(* IEC 61131-3 sources: axftcmlib/test, 13 files *)

(* ---- ActuatorTimeBasedTest.st ---- *)
USING Simatic.Ax.Commands;
USING Simatic.Ax.axftcmlib;
USING Simatic.Ax.IO.Output;
USING AxUnit.Assert;

NAMESPACE Simatic.Ax.axftcmlib

    {TestFixture}
    CLASS ActuatorTimeBasedTest
        VAR PROTECTED
            _actuator : ActuatorTimeBased;
            _actuatorStateLess : ActuatorTimeBased;
            _output : BinOutput;
            cmd : itfCommand;
            busy : BOOL;
        END_VAR

        {TestSetup}
        METHOD PUBLIC SetUp
            _actuator := _actuatorStateLess;
            _actuator.Q_ToWorkPosition := _output;
        END_METHOD

                {Test}
        METHOD PUBLIC TestTurnPneumaticCylinderPush_Expect_state_is_On
            cmd := _actuator.GoToWorkPosition();
            busy := cmd.Busy();
            AxUnit.Assert.Equal(expected := TRUE, actual := busy);
            AxUnit.Assert.Equal(expected := TRUE, actual := _output.IsOn());
            Equal(expected := TRUE, actual := _actuator.GetState() = ActuatorState#InWorkPosition);
        END_METHOD

        {Test}
        METHOD PUBLIC TestZylinderNotAsigned_Expected_ErrorFound_is_True
            VAR
                Test : BOOL;
            END_VAR
            _actuator.Q_ToWorkPosition := NULL;
            _actuator.Busy();
            AxUnit.Assert.Equal(Expected := TRUE, actual := _actuator.Error());
            ;
        END_METHOD

        {Test}
        METHOD PUBLIC TestPneumaticCylinderError_Expected_ErrorFound_TRUE
            VAR
                Test : BOOL;
            END_VAR

            Test := _actuator.Error();
            AxUnit.Assert.Equal(Expected := FALSE, actual := Test);
            ;
        END_METHOD

    END_CLASS

END_NAMESPACE

(* ---- Axis_Mock.st ---- *)
USING Simatic.Ax.IO.Input;
USING System.Timer;
USING Simatic.Ax.SimpleControlModules;

NAMESPACE Simatic.Ax.axftcmlib
    CLASS Axis_Mock
        IMPLEMENTS IAxis
        VAR PUBLIC
            State : PlcOpenState;
        END_VAR
        VAR PROTECTED

        END_VAR

        //-----------------------------------------
        // interface implementation
        METHOD PUBLIC MoveVelocity
            VAR_INPUT
                velocity : LREAL;
                direction : Direction;
            END_VAR
            ;
        END_METHOD
        METHOD PUBLIC MoveRelative : BOOL
            VAR_INPUT
                velocity : LREAL;
                distance : LINT;
            END_VAR
;
        END_METHOD
        METHOD PUBLIC MoveAbsolute : BOOL
            VAR_INPUT
                velocity : LREAL;
                position : LINT;
            END_VAR
;
        END_METHOD
        METHOD PUBLIC Homing : BOOL
            VAR_INPUT
                velocity : LREAL;
                direction : Direction;
            END_VAR
;
        END_METHOD
        METHOD PUBLIC Halt
            ;
        END_METHOD
        METHOD PUBLIC IsHomed : BOOL
            ;
        END_METHOD

        //-------------------------------------------------------------------------------
        // Section for private methods

        METHOD PUBLIC IsRunning : BOOL
            IsRunning := State = PlcOpenstate#Busy;
        END_METHOD

        METHOD PUBLIC Homing : BOOL
            VAR_INPUT
                Position : LINT;
            END_VAR

            ;
        END_METHOD
END_CLASS

END_NAMESPACE

(* ---- ColorSensor_test.st ---- *)
USING AxUnit.Assert;

NAMESPACE Simatic.Ax.axftcmlib
    {TestFixture}
    Class MyColorSensorTest

        VAR PROTECTED
            _testColorSensor : ColorSensor;
            //_testSubject : colors;
        END_VAR

        // METHOD PROTECTED SetUp
        //     _testColorSensor.OutputColor := _testSubject;
        // END_METHOD

        {Test}
        METHOD PUBLIC TestDetectionWhite_Expect_True
            VAR_TEMP
                Dummy : BOOL;
            END_VAR

            // THIS.SetUp();
            Dummy := FALSE;
            _testColorSensor.detectColor(DetectedColorValue := 9000);
            IF _testColorSensor.OutputColor = 1 THEN
                Dummy := TRUE;
            END_IF;
            AxUnit.Assert.Equal(expected := TRUE, actual := Dummy);
        END_METHOD

        {Test}
        METHOD PUBLIC TestDetectionRed_Expect_True
            VAR_TEMP
                Dummy : BOOL;
            END_VAR

            // THIS.SetUp();
            Dummy := FALSE;
            _testColorSensor.detectColor(DetectedColorValue := 14000);
            IF _testColorSensor.OutputColor = 2 THEN
                Dummy := TRUE;
            END_IF;
            AxUnit.Assert.Equal(expected := TRUE, actual := Dummy);
        END_METHOD

        {Test}
        METHOD PUBLIC TestDetectionBlue_Expect_True
            VAR_TEMP
                Dummy : BOOL;
            END_VAR

            // THIS.SetUp();
            Dummy := FALSE;
            _testColorSensor.detectColor(DetectedColorValue := 19000);
            IF _testColorSensor.OutputColor = 3 THEN
                Dummy := TRUE;
            END_IF;
            AxUnit.Assert.Equal(expected := TRUE, actual := Dummy);
        END_METHOD

    END_CLASS
END_NAMESPACE

(* ---- Compressor_test.st ---- *)
//USING Simatic.Ax.Cylinder;
USING AxUnit.Assert;
USING Simatic.Ax.IO.Input;
USING Simatic.Ax.axftcmlib;
USING Simatic.Ax.IO.Output;

NAMESPACE Simatic.Ax.axftcmlib
    {TestFixture}
    CLASS MyCompressorTest
        VAR PROTECTED
            _testCompressor : PneumaticCompressor;
            _testSubject : BinOutput;
        END_VAR
        METHOD PUBLIC  SetUp
            _testCompressor.ActiveCompressor := _testSubject;
        END_METHOD

        {Test}
        METHOD PUBLIC TestTurnCompressorOn_Expect_state_is_On
            THIS.SetUp();
            _testCompressor.PneumaticCompressorOn();
            AxUnit.Assert.Equal(expected := TRUE, actual :=_testSubject.IsOn()); // _testCompressor.ActiveCompressor.IsOn());
        END_METHOD

        {Test}
        METHOD PUBLIC TestTurnCompressorOff_Expect_state_is_Off
            THIS.SetUp();
            _testCompressor.PneumaticCompressorOff();
            AxUnit.Assert.Equal(expected := FALSE, actual := _testSubject.IsOn());
            END_METHOD

    END_CLASS
END_NAMESPACE

(* ---- Encoder_test.st ---- *)
USING Simatic.Ax.axftcmlib;

NAMESPACE Simatic.Ax.axftcmlib

    {TestFixture}
    CLASS MyEncoderTest
        VAR PROTECTED
            _testEncoderStatic : TimeBasedEncoder;
            _staticTimeProvider : TimeProviderMOCK_100ms_const;
            _staticAxis : Axis_Mock := (State := PlcOpenState#Busy);
        END_VAR

        METHOD PUBLIC SetUp
            VAR
                velocity : LREAL;
                dummyValue : INT;
            END_VAR
            dummyValue := 0;
            velocity := 1.0;
            _testEncoderStatic.velocity := 1.0;
            _testEncoderStatic.TimeProvider := _staticTimeProvider;
            _testEncoderStatic.EncoderAxis := _staticAxis;
            _testEncoderStatic.EncoderAxis.MoveVelocity(velocity, dummyvalue);
        END_METHOD

        {Test}
        METHOD PUBLIC TestPositionAfter100ms_Expect_position_equal
            THIS.SetUp();
            _testEncoderStatic.Reset();
            _testEncoderStatic.Evaluate();
            AxUnit.Assert.Equal(expected := 100, actual := _testEncoderStatic.GetValue());
            _testEncoderStatic.Evaluate();
            AxUnit.Assert.Equal(expected := 200, actual := _testEncoderStatic.GetValue());
            // Set Axis to stop
            _staticAxis.State := PlcOpenState#Done;
            _testEncoderStatic.Evaluate();
            AxUnit.Assert.Equal(expected := 200, actual := _testEncoderStatic.GetValue()); // dont integrate when axis is stopped
            // After Reset the GetValue should be 0
            _testEncoderStatic.Reset();
            AxUnit.Assert.Equal(expected := 0, actual := _testEncoderStatic.GetValue());

        END_METHOD
    END_CLASS

END_NAMESPACE

(* ---- test.st ---- *)
USING Simatic.Ax.IO.Input;
USING Simatic.Ax.Commands;
USING Simatic.Ax.axftcmlib;
USING Simatic.Ax.IO.Output;
USING AxUnit.Assert;

NAMESPACE Simatic.Ax.axftcmlib

    {TestFixture}
    CLASS TwoWayActuatorTest
        VAR PROTECTED
            _actuator : TwoWayActuator;
            _actuatorStateLess : TwoWayActuator;
            _qToWork : BinOutput;
            _qToHome : BinOutput;
            _outputStateLess : BinOutput;
            _iInHomePos : BinSignal;
            _iInWorkPos : BinSignal;
            _binSignalStateless : BinSignal;
            cmd : itfCommand;
            done : BOOL;
            busy : BOOL;
        END_VAR

        {TestSetup}
        METHOD PUBLIC SetUp
            _actuator := _actuatorStateLess;
            _actuator.Q_ToWorkPosition := _qToWork;
            _actuator.Q_ToHomePosition := _qToHome;
            _actuator.I_InHomePosition := _iInHomePos;
            _actuator.I_InWorkPosition := _iInWorkPos;
            _iInHomePos := _binSignalStateless;
            _iInWorkPos := _binSignalStateless;
            _qToWork := _outputStateLess;
            _qToHome := _outputStateLess;
            busy := FALSE;
            cmd := NULL;
        END_METHOD

        {Test}
        METHOD PUBLIC GoToWorkPosition_Swiches_Q_ToWorkPosition_On_And_Returns_Busy
            cmd := _actuator.GoToWorkPosition();
            busy := cmd.Busy();
            AxUnit.Assert.Equal(expected := TRUE, actual := busy);
            AxUnit.Assert.Equal(expected := TRUE, actual := _qToWork.IsOn());
            AxUnit.Assert.Equal(expected := FALSE, actual := _qToHome.IsOn());
            Equal(expected := TRUE, actual := _actuator.GetState() = ActuatorState#MoveToWorkPosition);
        END_METHOD

        {Test}
        METHOD PUBLIC GoToWorkPosition_Returns_Done_When_end_position_is_already_reached
            _iInWorkPos.ReadCyclic(signal := TRUE);
            cmd := _actuator.GoToWorkPosition();
            busy := cmd.Busy();
            IF NOT(busy) THEN
                done := cmd.Done();
            END_IF;
            AxUnit.Assert.Equal(expected := FALSE, actual := busy);
            AxUnit.Assert.Equal(expected := TRUE, actual := done);
            AxUnit.Assert.Equal(expected := FALSE, actual := _qToWork.IsOn());
            AxUnit.Assert.Equal(expected := FALSE, actual := _qToHome.IsOn());
            Equal(expected := TRUE, actual := _actuator.GetState() = ActuatorState#InWorkPosition);
        END_METHOD

        {Test}
        METHOD PUBLIC Reaching_WorkPosition_Switches_Q_ToWorkPosition_Off_And_Returns_Done
            THIS.GoToWorkPosition_Swiches_Q_ToWorkPosition_On_And_Returns_Busy();
            _iInWorkPos.ReadCyclic(signal := TRUE);
            busy := cmd.Busy();
            IF NOT(busy) THEN
                done := cmd.Done();
            END_IF;
            AxUnit.Assert.Equal(expected := FALSE, actual := busy);
            AxUnit.Assert.Equal(expected := TRUE, actual := done);
            AxUnit.Assert.Equal(expected := FALSE, actual := _qToWork.IsOn());
            AxUnit.Assert.Equal(expected := FALSE, actual := _qToHome.IsOn());
            Equal(expected := TRUE, actual := _actuator.GetState() = ActuatorState#InWorkPosition);
        END_METHOD

        // Test Home Position
        {Test}
        METHOD PUBLIC GoToHomePosition_Swiches_Q_ToHomePosition_On_And_Returns_Busy
            cmd := _actuator.GoToHomePosition();
            busy := cmd.Busy();
            AxUnit.Assert.Equal(expected := TRUE, actual := busy);
            AxUnit.Assert.Equal(expected := FALSE, actual := _qToWork.IsOn());
            AxUnit.Assert.Equal(expected := TRUE, actual := _qToHome.IsOn());
            Equal(expected := TRUE, actual := _actuator.GetState() = ActuatorState#MoveToHomePosition);
        END_METHOD

        {Test}
        METHOD PUBLIC GoToHomePosition_Returns_Done_When_end_position_is_already_reached
            _iInHomePos.ReadCyclic(signal := TRUE);
            cmd := _actuator.GoToHomePosition();
            busy := cmd.Busy();
            IF NOT(busy) THEN
                done := cmd.Done();
            END_IF;
            AxUnit.Assert.Equal(expected := FALSE, actual := busy);
            AxUnit.Assert.Equal(expected := TRUE, actual := done);
            AxUnit.Assert.Equal(expected := FALSE, actual := _qToWork.IsOn());
            AxUnit.Assert.Equal(expected := FALSE, actual := _qToHome.IsOn());
            Equal(expected := TRUE, actual := _actuator.GetState() = ActuatorState#InHomePosition);
        END_METHOD

        {Test}
        METHOD PUBLIC Reaching_HomePosition_Switches_Q_ToHomePosition_Off_And_Returns_Done
            THIS.GoToHomePosition_Swiches_Q_ToHomePosition_On_And_Returns_Busy();
            _iInHomePos.ReadCyclic(signal := TRUE);
            busy := cmd.Busy();
            IF NOT(busy) THEN
                done := cmd.Done();
            END_IF;
            AxUnit.Assert.Equal(expected := FALSE, actual := busy);
            AxUnit.Assert.Equal(expected := TRUE, actual := done);
            AxUnit.Assert.Equal(expected := FALSE, actual := _qToWork.IsOn());
            AxUnit.Assert.Equal(expected := FALSE, actual := _qToHome.IsOn());
            Equal(expected := TRUE, actual := _actuator.GetState() = ActuatorState#InHomePosition);
        END_METHOD
    END_CLASS

END_NAMESPACE

(* ---- TestAxis.st ---- *)
USING Simatic.Ax.IO.Output;
USING Simatic.Ax.IO.Input;
USING Simatic.Ax.axftcmlib;
USING AxUnit.Assert;

// USING Simatic.Ax.SimpleControlModules;
NAMESPACE Simatic.Ax.Library

    {TestFixture}
    CLASS TestAxisHoming
        VAR PROTECTED
            _axis : Axis;
            _refSwitch : BinSignal;
            _motor : MotorFT;
            _fwd : BinOutput;
            _rvs : BinOutput;
            _encoder : Simatic.Ax.SimpleControlModules.EncoderAB;
        END_VAR
        METHOD PUBLIC Setup
            _motor.Forward := _fwd;
            _motor.Reverse := _rvs;
            _axis.Motor := _motor;
            _axis.Encoder := _encoder;
            _axis.ReferenceSwitch := _refSwitch;
        END_METHOD
        {Test}
        METHOD PUBLIC TestForwardDirection_Expect_Fwd_IsOn
            THIS.Setup();
            _axis.MoveVelocity(direction := Direction#Forward);
            _axis.RunCyclic();
            Equal(expected := TRUE, actual := _axis.GetPlcOpenState() = PlcOpenState#Busy);
            Equal(expected := TRUE, actual := _fwd.IsOn());
            Equal(expected := FALSE, actual := _rvs.IsOn());
        END_METHOD
        {Test}
        METHOD PUBLIC Homing_from_outside_of_the_referecne_sensor_Move_reverse
            THIS.Setup();
            _axis.Homing(direction := Direction#Reverse);
            _axis.RunCyclic();
            Equal(expected := TRUE, actual := _axis.GetPlcOpenState() = PlcOpenState#Busy);
            _axis.RunCyclic();
            Equal(expected := FALSE, actual := _fwd.IsOn());
            Equal(expected := TRUE, actual := _rvs.IsOn());
        END_METHOD

        {Test}
        METHOD PUBLIC Homing_from_outside_of_the_referecne_sensor_Move_forward
            THIS.Setup();
            _axis.Homing(direction := Direction#Forward);
            _axis.RunCyclic();
            Equal(expected := TRUE, actual := _axis.GetPlcOpenState() = PlcOpenState#Busy);
            _axis.RunCyclic();
            Equal(expected := TRUE, actual := _fwd.IsOn());
            Equal(expected := FALSE, actual := _rvs.IsOn());
        END_METHOD

        {Test}
        METHOD PUBLIC Homing_untilsensor_has_reached
            VAR_TEMP
                isHomed : BOOL;
            END_VAR
            THIS.Setup();

            _axis.Homing(direction := Direction#Forward);
            _axis.RunCyclic();

            _refSwitch.ReadCyclic(signal := FALSE);
            _axis.RunCyclic();
            Equal(expected := TRUE, actual := _axis.GetPlcOpenState() = PlcOpenState#Busy);
            Equal(expected := FALSE, actual := _axis.GetPlcOpenState() = PlcOpenState#Error);
            Equal(expected := FALSE, actual := _axis.GetPlcOpenState() = PlcOpenState#Done);
            Equal(expected := TRUE, actual := _fwd.IsOn());
            Equal(expected := FALSE, actual := _rvs.IsOn());

            _refSwitch.ReadCyclic(signal := FALSE);
            _axis.RunCyclic();
            Equal(expected := TRUE, actual := _axis.GetPlcOpenState() = PlcOpenState#Busy);
            Equal(expected := FALSE, actual := _axis.GetPlcOpenState() = PlcOpenState#Error);
            Equal(expected := FALSE, actual := _axis.GetPlcOpenState() = PlcOpenState#Done);
            Equal(expected := TRUE, actual := _fwd.IsOn());
            Equal(expected := FALSE, actual := _rvs.IsOn());

            _refSwitch.ReadCyclic(signal := FALSE);
            _axis.RunCyclic();
            Equal(expected := TRUE, actual := _axis.GetPlcOpenState() = PlcOpenState#Busy);
            Equal(expected := FALSE, actual := _axis.GetPlcOpenState() = PlcOpenState#Error);
            Equal(expected := FALSE, actual := _axis.GetPlcOpenState() = PlcOpenState#Done);
            Equal(expected := TRUE, actual := _fwd.IsOn());
            Equal(expected := FALSE, actual := _rvs.IsOn());

            _refSwitch.ReadCyclic(signal := TRUE);
            _axis.RunCyclic();
            _axis.RunCyclic();
            Equal(expected := FALSE, actual := _axis.GetPlcOpenState() = PlcOpenState#Busy);
            Equal(expected := FALSE, actual := _axis.GetPlcOpenState() = PlcOpenState#Error);
            Equal(expected := TRUE, actual := _axis.GetPlcOpenState() = PlcOpenState#Done);
            Equal(expected := FALSE, actual := _fwd.IsOn());
            Equal(expected := FALSE, actual := _rvs.IsOn());
            Equal(expected := TRUE, actual := _axis.IsHomed());
        END_METHOD

    END_CLASS

END_NAMESPACE

(* ---- TestAxisManualHoming.st ---- *)
USING Simatic.Ax.IO.Output;
USING Simatic.Ax.IO.Input;
USING Simatic.Ax.axftcmlib;
USING AxUnit.Assert;

// USING Simatic.Ax.SimpleControlModules;
NAMESPACE Simatic.Ax.Library

    {TestFixture}
    CLASS TestAxisManualHoming
        VAR PROTECTED
            _axis : Axis;
            _refSwitch : BinSignal;
            _motor : MotorFT;
            _fwd : BinOutput;
            _rvs : BinOutput;
            _encoder : Simatic.Ax.SimpleControlModules.EncoderAB;
        END_VAR
        METHOD PUBLIC Setup
            _motor.Forward := _fwd;
            _motor.Reverse := _rvs;
            _axis.Motor := _motor;
            _axis.Encoder := _encoder;
            _axis.ReferenceSwitch := _refSwitch;
        END_METHOD
        {Test}
        METHOD PUBLIC AxisReturnes_IsHomed_when_Homing_Method_isCalled
            THIS.Setup();
            Equal(expected := FALSE, actual := _axis.IsHomed());
            _axis.Homing(position := 100);
            Equal(expected := TRUE, actual := _axis.IsHomed());
            Equal(expected := TRUE, actual := _axis.GetPlcOpenState() = PlcOpenState#Done);
            _axis.RunCyclic();
            Equal(expected := FALSE, actual := _axis.GetPlcOpenState() = PlcOpenState#Done);
        END_METHOD
    END_CLASS

END_NAMESPACE

(* ---- TestAxisMoveAbsolut.st ---- *)
USING Simatic.Ax.IO.Output;
USING Simatic.Ax.IO.Input;
USING Simatic.Ax.axftcmlib;
USING AxUnit.Assert;

// USING Simatic.Ax.SimpleControlModules;
NAMESPACE Simatic.Ax.Library

    {TestFixture}
    CLASS TestAxisMoveAbsolut
        VAR PROTECTED
            _axis : Axis;
            _refSwitch : BinSignal;
            _motor : MotorFT;
            _fwd : BinOutput;
            _rvs : BinOutput;
            _encoder : Simatic.Ax.SimpleControlModules.EncoderAB;
        END_VAR
        METHOD PUBLIC Setup
            _motor.Forward := _fwd;
            _motor.Reverse := _rvs;
            _axis.Motor := _motor;
            _axis.Encoder := _encoder;
            _axis.ReferenceSwitch := _refSwitch;
        END_METHOD
        METHOD PUBLIC Home : BOOL
            VAR_INPUT
                axis : REF_TO Axis;
                refSwitch : REF_TO BinSignal;
            END_VAR
            axis^.Homing(direction := Direction#Forward);
            refSwitch^.ReadCyclic(signal := FALSE);
            axis^.RunCyclic();
            refSwitch^.ReadCyclic(signal := TRUE);
            axis^.RunCyclic();
            // one additional cycle to finalize the Homing
            axis^.RunCyclic();
            Home := axis^.IsHomed();
        END_METHOD
        {Test}
        METHOD PUBLIC Test_MoveAbsolut_on_a_not_homed_axis_which_results_in_an_error
            VAR_TEMP
                isHomed : BOOL;
            END_VAR
            THIS.Setup();
            _axis.MoveAbsolute(velocity := 100.0, position := LINT#100);
            _axis.RunCyclic();
            Equal(expected := FALSE, actual := _axis.GetPlcOpenState() = PlcOpenState#Busy);
            Equal(expected := TRUE, actual := _axis.GetPlcOpenState() = PlcOpenState#Error);
            Equal(expected := FALSE, actual := _axis.GetPlcOpenState() = PlcOpenState#Done);
        END_METHOD
        {Test}
        METHOD PUBLIC Test_MoveAbsolut_on_a_homed_axis
            VAR_TEMP
                isHomed : BOOL;
            END_VAR
            THIS.Setup();
            isHomed := THIS.Home(axis := REF(_axis), refSwitch := REF(_refSwitch));
            Equal(expected := TRUE, actual := isHomed);
            Equal(expected := FALSE, actual := _fwd.IsOn());
            Equal(expected := FALSE, actual := _rvs.IsOn());
            // start Axis to move to position 100
            _axis.MoveAbsolute(velocity := 100.0, position := LINT#100);
            _axis.RunCyclic();
            Equal(expected := TRUE, actual := _axis.GetPlcOpenState() = PlcOpenState#Busy);
            Equal(expected := FALSE, actual := _axis.GetPlcOpenState() = PlcOpenState#Error);
            Equal(expected := FALSE, actual := _axis.GetPlcOpenState() = PlcOpenState#Done);
            Equal(expected := TRUE, actual := _fwd.IsOn());
            Equal(expected := FALSE, actual := _rvs.IsOn());
            // Axis is at position 99
            _encoder.SetValue(value := LINT#99);
            _axis.RunCyclic();
            Equal(expected := TRUE, actual := _axis.GetPlcOpenState() = PlcOpenState#Busy);
            // test axis in position
            _encoder.SetValue(value := LINT#100);
            _axis.RunCyclic();
            _axis.RunCyclic();
            Equal(expected := TRUE, actual := _axis.GetPlcOpenState() = PlcOpenState#Done);
            Equal(expected := FALSE, actual := _axis.GetPlcOpenState() = PlcOpenState#Busy);
            Equal(expected := FALSE, actual := _fwd.IsOn());
            Equal(expected := FALSE, actual := _rvs.IsOn());            // test axis in position - done after one cycle is false
            _encoder.SetValue(value := LINT#100);
            _axis.RunCyclic();
            Equal(expected := FALSE, actual := _axis.GetPlcOpenState() = PlcOpenState#Done);
            Equal(expected := FALSE, actual := _axis.GetPlcOpenState() = PlcOpenState#Busy);
        END_METHOD
        {Test}
        METHOD PUBLIC Move_Absolut_on_a_axis_which_is_already_inPos
            VAR_TEMP
                isHomed : BOOL;
            END_VAR
            THIS.Setup();
            isHomed := THIS.Home(axis := REF(_axis), refSwitch := REF(_refSwitch));
            Equal(expected := TRUE, actual := isHomed);
            Equal(expected := FALSE, actual := _fwd.IsOn());
            Equal(expected := FALSE, actual := _rvs.IsOn());
            // start Axis to move to position 100
            _encoder.SetValue(value := LINT#100);
            _axis.MoveAbsolute(velocity := 100.0, position := LINT#100);
            _axis.RunCyclic();
            Equal(expected := FALSE, actual := _axis.GetPlcOpenState() = PlcOpenState#Busy);
            Equal(expected := FALSE, actual := _axis.GetPlcOpenState() = PlcOpenState#Error);
            Equal(expected := TRUE, actual := _axis.GetPlcOpenState() = PlcOpenState#Done);
            Equal(expected := FALSE, actual := _fwd.IsOn());
            Equal(expected := FALSE, actual := _rvs.IsOn());
        END_METHOD
    END_CLASS

END_NAMESPACE

(* ---- TestMoveVelocity.st ---- *)
USING Simatic.Ax.IO.Output;
USING Simatic.Ax.IO.Input;
USING Simatic.Ax.axftcmlib;
USING AxUnit.Assert;

// USING Simatic.Ax.SimpleControlModules;
NAMESPACE Simatic.Ax.Library

    {TestFixture}
    CLASS TestMoveVelocity
        VAR PROTECTED
            _axis : Axis;
            _refSwitch : BinSignal;
            _motor : MotorFT;
            _fwd : BinOutput;
            _rvs : BinOutput;
            _encoder : Simatic.Ax.SimpleControlModules.EncoderAB;
        END_VAR
        METHOD PUBLIC Setup
            _motor.Forward := _fwd;
            _motor.Reverse := _rvs;
            _axis.Motor := _motor;
            _axis.Encoder := _encoder;
            _axis.ReferenceSwitch := _refSwitch;
        END_METHOD
        {Test}
        METHOD PUBLIC MotorForward_IsOn_When_MoveVelocityIsCalled_With_Direction_Forward
            THIS.Setup();
            _axis.MoveVelocity(direction := Direction#Forward);
            _axis.RunCyclic();
            Equal(expected := TRUE, actual := _fwd.IsOn());
            Equal(expected := FALSE, actual := _rvs.IsOn());
            Equal(expected := TRUE, actual := _axis.GetPlcOpenState() = PlcOpenState#Busy);
        END_METHOD
        {Test}
        METHOD PUBLIC MotorReverse_IsOn_When_MoveVelocityIsCalled_With_Direction_Reverse
            THIS.Setup();
            _axis.MoveVelocity(direction := Direction#Reverse);
            _axis.RunCyclic();
            Equal(expected := FALSE, actual := _fwd.IsOn());
            Equal(expected := TRUE, actual := _rvs.IsOn());
            Equal(expected := TRUE, actual := _axis.GetPlcOpenState() = PlcOpenState#Busy);
        END_METHOD
        {Test}
        METHOD PUBLIC A_Moving_AxisStops_OnHalt;
            THIS.MotorForward_IsOn_When_MoveVelocityIsCalled_With_Direction_Forward();
            _axis.Halt();
            Equal(expected := FALSE, actual := _fwd.IsOn());
            Equal(expected := FALSE, actual := _rvs.IsOn());
            Equal(expected := TRUE, actual := _axis.GetPlcOpenState() = PlcOpenState#Done);
            _axis.RunCyclic();
            Equal(expected := FALSE, actual := _axis.GetPlcOpenState() = PlcOpenState#Done);
        END_METHOD
    END_CLASS

END_NAMESPACE

(* ---- TimeBasedActuatorTest.st ---- *)
USING Simatic.Ax.Commands;
USING Simatic.Ax.axftcmlib;
USING Simatic.Ax.IO.Output;
USING AxUnit.Assert;

NAMESPACE Simatic.Ax.axftcmlib

    {TestFixture}
    CLASS TimeBasedActuatorTest
        VAR PROTECTED
            _actuator : TimeBasedActuator;
            _actuatorStateLess : TimeBasedActuator;
            _output : BinOutput;
            cmd : itfCommand;
            busy : BOOL;
        END_VAR

        {TestSetup}
        METHOD PUBLIC SetUp
            _actuator := _actuatorStateLess;
            _actuator.Q_ToWorkPosition := _output;
        END_METHOD

                {Test}
        METHOD PUBLIC TestTurnPneumaticCylinderPush_Expect_state_is_On
            cmd := _actuator.GoToWorkPosition();
            busy := cmd.Busy();
            AxUnit.Assert.Equal(expected := TRUE, actual := busy);
            AxUnit.Assert.Equal(expected := TRUE, actual := _output.IsOn());
            Equal(expected := TRUE, actual := _actuator.GetState() = ActuatorState#InWorkPosition);
        END_METHOD

        {Test}
        METHOD PUBLIC TestZylinderNotAsigned_Expected_ErrorFound_is_True
            VAR
                Test : BOOL;
            END_VAR
            _actuator.Q_ToWorkPosition := NULL;
            _actuator.Busy();
            AxUnit.Assert.Equal(Expected := TRUE, actual := _actuator.Error());
            ;
        END_METHOD

        {Test}
        METHOD PUBLIC TestPneumaticCylinderError_Expected_ErrorFound_TRUE
            VAR
                Test : BOOL;
            END_VAR

            Test := _actuator.Error();
            AxUnit.Assert.Equal(Expected := FALSE, actual := Test);
            ;
        END_METHOD

    END_CLASS

END_NAMESPACE

(* ---- Timeprovider_Mock.st ---- *)
NAMESPACE Simatic.Ax.axftcmlib
/// Mock for a ITimePrivider wich returns always 100ms.
    CLASS TimeProviderMOCK_100ms_const
        IMPLEMENTS ITimeprovider

        METHOD PUBLIC GetElapsedSeconds : LREAL
         GetElapsedSeconds := 0.1;
        END_METHOD
    END_CLASS

END_NAMESPACE

(* ---- TwoWayActuatorTest.st ---- *)
USING Simatic.Ax.IO.Input;
USING Simatic.Ax.Commands;
USING Simatic.Ax.axftcmlib;
USING Simatic.Ax.IO.Output;
USING AxUnit.Assert;

NAMESPACE Simatic.Ax.axftcmlib

    {TestFixture}
    CLASS TwoWayActuatorTest
        VAR PROTECTED
            _actuator : TwoWayActuator;
            _actuatorStateLess : TwoWayActuator;
            _qToWork : BinOutput;
            _qToHome : BinOutput;
            _outputStateLess : BinOutput;
            _iInHomePos : BinSignal;
            _iInWorkPos : BinSignal;
            _binSignalStateless : BinSignal;
            cmd : itfCommand;
            done : BOOL;
            busy : BOOL;
        END_VAR

        {TestSetup}
        METHOD PUBLIC SetUp
            _actuator := _actuatorStateLess;
            _actuator.Q_ToWorkPosition := _qToWork;
            _actuator.Q_ToHomePosition := _qToHome;
            _actuator.I_InHomePosition := _iInHomePos;
            _actuator.I_InWorkPosition := _iInWorkPos;
            _iInHomePos := _binSignalStateless;
            _iInWorkPos := _binSignalStateless;
            _qToWork := _outputStateLess;
            _qToHome := _outputStateLess;
            busy := FALSE;
            cmd := NULL;
        END_METHOD

        {Test}
        METHOD PUBLIC GoToWorkPosition_Swiches_Q_ToWorkPosition_On_And_Returns_Busy
            cmd := _actuator.GoToWorkPosition();
            busy := cmd.Busy();
            AxUnit.Assert.Equal(expected := FALSE, actual := busy);
            AxUnit.Assert.Equal(expected := TRUE, actual := _qToWork.IsOn());
            AxUnit.Assert.Equal(expected := FALSE, actual := _qToHome.IsOn());
            Equal(expected := TRUE, actual := _actuator.GetState() = ActuatorState#MoveToWorkPosition);
        END_METHOD

        {Test}
        METHOD PUBLIC GoToWorkPosition_Returns_Done_When_end_position_is_already_reached
            _iInWorkPos.ReadCyclic(signal := TRUE);
            cmd := _actuator.GoToWorkPosition();
            busy := cmd.Busy();
            IF NOT(busy) THEN
                done := cmd.Done();
            END_IF;
            AxUnit.Assert.Equal(expected := FALSE, actual := busy);
            AxUnit.Assert.Equal(expected := TRUE, actual := done);
            AxUnit.Assert.Equal(expected := FALSE, actual := _qToWork.IsOn());
            AxUnit.Assert.Equal(expected := FALSE, actual := _qToHome.IsOn());
            Equal(expected := TRUE, actual := _actuator.GetState() = ActuatorState#InWorkPosition);
        END_METHOD

        // {Test}
        // METHOD PUBLIC Reaching_WorkPosition_Switches_Q_ToWorkPosition_Off_And_Returns_Done
        //     THIS.GoToWorkPosition_Swiches_Q_ToWorkPosition_On_And_Returns_Busy();
        //     _iInWorkPos.ReadCyclic(signal := TRUE);
        //     busy := cmd.Busy();
        //     IF NOT(busy) THEN
        //         done := cmd.Done();
        //     END_IF;
        //     AxUnit.Assert.Equal(expected := FALSE, actual := busy);
        //     AxUnit.Assert.Equal(expected := TRUE, actual := done);
        //     AxUnit.Assert.Equal(expected := FALSE, actual := _qToWork.IsOn());
        //     AxUnit.Assert.Equal(expected := FALSE, actual := _qToHome.IsOn());
        //     Equal(expected := TRUE, actual := _actuator.GetState() = ActuatorState#InWorkPosition);
        // END_METHOD

        // // Test Home Position
        // {Test}
        // METHOD PUBLIC GoToHomePosition_Swiches_Q_ToHomePosition_On_And_Returns_Busy
        //     cmd := _actuator.GoToHomePosition();
        //     busy := cmd.Busy();
        //     AxUnit.Assert.Equal(expected := TRUE, actual := busy);
        //     AxUnit.Assert.Equal(expected := FALSE, actual := _qToWork.IsOn());
        //     AxUnit.Assert.Equal(expected := TRUE, actual := _qToHome.IsOn());
        //     Equal(expected := TRUE, actual := _actuator.GetState() = ActuatorState#MoveToHomePosition);
        // END_METHOD

        // {Test}
        // METHOD PUBLIC GoToHomePosition_Returns_Done_When_end_position_is_already_reached
        //     _iInHomePos.ReadCyclic(signal := TRUE);
        //     cmd := _actuator.GoToHomePosition();
        //     busy := cmd.Busy();
        //     IF NOT(busy) THEN
        //         done := cmd.Done();
        //     END_IF;
        //     AxUnit.Assert.Equal(expected := FALSE, actual := busy);
        //     AxUnit.Assert.Equal(expected := TRUE, actual := done);
        //     AxUnit.Assert.Equal(expected := FALSE, actual := _qToWork.IsOn());
        //     AxUnit.Assert.Equal(expected := FALSE, actual := _qToHome.IsOn());
        //     Equal(expected := TRUE, actual := _actuator.GetState() = ActuatorState#InHomePosition);
        // END_METHOD

        // {Test}
        // METHOD PUBLIC Reaching_HomePosition_Switches_Q_ToHomePosition_Off_And_Returns_Done
        //     THIS.GoToHomePosition_Swiches_Q_ToHomePosition_On_And_Returns_Busy();
        //     _iInHomePos.ReadCyclic(signal := TRUE);
        //     busy := cmd.Busy();
        //     IF NOT(busy) THEN
        //         done := cmd.Done();
        //     END_IF;
        //     AxUnit.Assert.Equal(expected := FALSE, actual := busy);
        //     AxUnit.Assert.Equal(expected := TRUE, actual := done);
        //     AxUnit.Assert.Equal(expected := FALSE, actual := _qToWork.IsOn());
        //     AxUnit.Assert.Equal(expected := FALSE, actual := _qToHome.IsOn());
        //     Equal(expected := TRUE, actual := _actuator.GetState() = ActuatorState#InHomePosition);
        // END_METHOD
    END_CLASS

END_NAMESPACE
